{attribute addProperty BoxType "EL1259-0000-0016"}
{attribute addProperty Id "StatusAT %I*Status_32B8CA6210913.625"}
{attribute addProperty CRC "1523873199"}
{attribute addProperty SizeInBites "109"}
{attribute addProperty SizeInBytes "13.625"}
TYPE MTO_Inputs_Channel_5AD475AF :
STRUCT
	{attribute addProperty Name "Status"}
	Status AT %I* : Status_32B8CA62;
END_STRUCT
END_TYPE

(* stored: Version 1.2.0.0, ProductVersion 3.1.4024.9
   DUT MTO_Inputs_Channel_5AD475AF: Id {b52e9e0e-6afb-4256-9e2a-a7df712a98ca} *)
